// TIA Portal V20 export
FUNCTION_BLOCK "FB_CycleStartStop"   // FB406, SCL
{ S7_Optimized_Access := 'TRUE' }
// stored: AutoNumber false, MemoryReserve 100, SetENOAutomatically false
   VAR
      sChan1Start : Bool;
      sResquestStopNextCycle : Bool;
      sTimePowerSupplyAlarm : TON_TIME;
      sRT_CNAskStopCycle : R_TRIG;
   END_VAR
   VAR CONSTANT
      TIME_POWER_SUPPPLY_ALARM : Time := T#5s;
   END_VAR
BEGIN
   REGION Description header 
       //==================================================================================
       // POSALUX Swiss SA / (C) Copyright 2024
       //----------------------------------------------------------------------------------
       // Title: Start and stop cycle
       // Comment/Function:  Replacement of the Siemens standard cycle stop button with a
       // customized method for stopping and restarting the cycle, adabted to the specific
       // needs of the application.
       // 
       // Author: Gowsigan SRITHARAN
       // Engineering: TIA Portal v17
       //----------------------------------------------------------------------------------
       // Change log table:
       // Version  | Date     | Expert in charge | Changes applied
       // ---------|----------|------------------|------------------------------------
       // 00.00.01 | 20241202 | GSR              | First released version
       // ==================================================================================
   END_REGION

   REGION Start memo
       // Start channel
       IF "LBP_Chan1".E_ProgRunning THEN
           #sChan1Start := TRUE;
       END_IF;

       // Reset channel
       IF "LBP_Chan1".E_ChanReset THEN
           #sChan1Start := FALSE;
       END_IF;
   END_REGION

   REGION Start disabled
       "LBP_Chan1".A_NCStartDisabl :="DB_Alarms".sAlarmsLevel3 OR "DB_Alarms".sAlarmsLevel4 OR "DB_Alarms".sAlarmsLevel5 OR  "DB_Alarms".sAlarmsLevel6;
       "LBP_Chan1".A_NCStart := ("MCP1_In".cycleStart OR "DB_HMISetting".StartAutoReq) AND (NOT"LBP_Chan1".A_NCStartDisabl);

       "DB_HMISetting".StartAutoReq := FALSE;
   END_REGION

   REGION Mode change disabled
       "LBP_ModeGroup".A_MCDisable := #sChan1Start AND NOT "LBP_Chan1".E_M01;    // Disable change CNC mode
   END_REGION

   REGION  Stop request (From MCP or alarms)
       // If key stop cycle is pressed or alarm level3 then request stop
       IF #sChan1Start
           AND (NOT "MCP1_In".cycleStop OR "DB_HMISetting".StopAutoReq OR "DB_Alarms".sAlarmsLevel3 OR "DB_Alarms".sAlarmsLevel4) THEN
           #sResquestStopNextCycle := TRUE;
           "LBP_AlarmMsgs".UserA[00].A70UUxx[60] := TRUE; // Msg "Stop program requested by operator"

           "DB_HMISetting".StopAutoReq := FALSE;
       END_IF;
   END_REGION

   REGION Wait Channel stopped
       IF  #sResquestStopNextCycle AND "LBP_Chan1".E_M01 THEN
           #sResquestStopNextCycle := FALSE;
       END_IF;
   END_REGION

   REGION Reset stop at next step
       IF "LBP_Chan1".MDyn[78] OR "LBP_Chan1".E_ChanReset THEN // M78 ISO command to restart 
           "LBP_NC".A_Set_Inp31 := FALSE;
           "LBP_AlarmMsgs".UserA[0].A70UUxx[60] := FALSE;
           #sResquestStopNextCycle := FALSE;
       END_IF;
   END_REGION

   REGION LED NC Start / Stop
       // Stop LED
       "MCP1_Out".LEDcycleStop :=
       NOT "LBP_Chan1".E_ChanReset
       AND NOT "LBP_Chan1".A_Ref
       AND ("LBP_Chan1".E_ProgStop
       OR "LBP_Chan1".E_ProgInterrupt
       OR "LBP_Chan1".E_ProgAborted) OR
       (#sResquestStopNextCycle AND "Clock_1Hz");

       // Start LED
       "MCP1_Out".LEDcycleStart :="LBP_Chan1".E_ProgRunning OR "LBP_Chan1".A_Ref;

      // Cycle start LED (Key [19])
       "DB_McpKeyboardSignals".sStartCycle.sLedSWStatus := "LBP_Chan1".E_ProgRunning OR "LBP_Chan1".A_Ref;
   END_REGION

   REGION Channel feed disable (Power Supply error)
       #sTimePowerSupplyAlarm(IN := "DB_PowerOn".sMachinePower
                              AND (NOT "DB_DigitalInputs".sPowerReady.sSWStatus
                              OR NOT "DB_DigitalInputs".sAlarmI2T.sSWStatus),
                              PT := #TIME_POWER_SUPPPLY_ALARM);

       IF #sTimePowerSupplyAlarm.Q THEN
           "LBP_AlarmMsgs".Chan[1].FDD[1] := TRUE;
       ELSIF "DB_McpKeyboardSignals".sAlarmReset.sKeySWStatus THEN
           "LBP_AlarmMsgs".Chan[1].FDD[1] := FALSE;
       END_IF;

       IF #sTimePowerSupplyAlarm.Q AND NOT "DB_DigitalInputs".sPowerReady.sSWStatus THEN
           "LBP_AlarmMsgs".UserA[03].A70UUxx[30] := TRUE;       // Msg: 700330 "Drives power supply not ready"
       END_IF;

       IF #sTimePowerSupplyAlarm.Q AND NOT "DB_DigitalInputs".sAlarmI2T.sSWStatus THEN
           "LBP_AlarmMsgs".UserA[03].A70UUxx[31] := TRUE;       // Msg: 700331 "Drives power supply overload"
       END_IF;
   END_REGION
END_FUNCTION_BLOCK
